(* Schneider Machine Expert - Basic project p9, file version 1.8.0.0 *)
(* ProjectInformations: Name=New project *)

HARDWARE
  Cpu 0: TM221CE16R
  EthernetConfiguration: NetworkName=M221, IpAllocationMode=FixedAddress, IpAddress=192.168.162.202, SubnetMask=255.255.255.0
  SerialLineConfiguration: Baud=Baud19200, Parity=ParityEven, DataBits=DataBits8, StopBits=StopBits1, PhysicalMedium=PhysicalMediumRs485, TransmissionMode=TransmissionModeModbusRtu, SlaveId=1, Addressing=SlaveAddressing
  MastTask: UsePeriodScanMode=false, PeriodScan=100
  FastTask: Period=255
  CpuBehavior: StartingMode=StartAsPreviousState, AutoSaveRamOnEeprom=true, WatchdogPeriod=250

SYMBOLS  (address, symbol, comment, settings)
  %TM0        [Preset=3, Base=OneSecond, IsRetentive=true]

POU New POU
  (* SectionNumber=1 *)

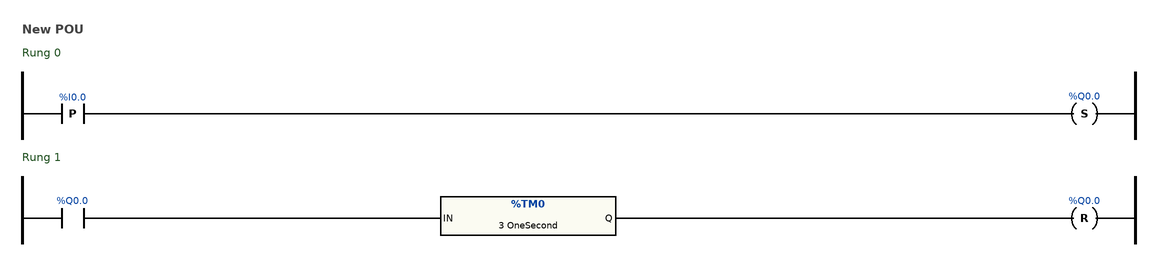

// Rung 0
  LDR %I0.0
  S %Q0.0
  // as ST:
  //   IF RISING(%I0.0) THEN %Q0.0 := TRUE; END_IF;

// Rung 1
  BLK %TM0
  LD %Q0.0
  IN
  OUT_BLK
  LD Q
  R %Q0.0
  END_BLK
  // as ST:
  //   %TM0(IN := %Q0.0);
  //   IF %TM0.Q THEN %Q0.0 := FALSE; END_IF;
